# EPICS substitutions: ssaApp/Db/ssa1.substitutions
# asyn record for the underlying asyn octet port
#file "ASYN/db/asynRecord.db" { pattern
#{P,           R,       PORT,      ADDR,   IMAX,    OMAX}
#{SSA1:    OctetAsyn,   ssa1,        0,      125,      123}
#}

# These are the B0 outputs done with bit access.
file "bo_word.template"
{ pattern
{P,           R,        PORT,      OFFSET,   MASK,	ZNAM,  ONAM}
{SSA1:,    OUT1,        RF1_Out_Word,    0,     0x0001,	0, 	1}
{SSA1:,    OUT2,        RF1_Out_Word,    1,     0x0001,	0,	1}
{SSA1:,    OUT4,        RF1_Out_Word,    3,     0x0001,	0,	1}
{SSA1:,    OUT5,        RF1_Out_Word,    4,     0x0001,	0,	1}
{SSA1:,	   OUT6,	RF1_Out_Word,    5,     0x0001,	0,	1}
}

# These are the A0 ouput donw with word write
file "longout.template"
{ pattern
{P,           R,        PORT,      OFFSET}
{SSA1:,    OUT3,        RF1_Out_Word,    2}
}

# There are the Inputs done with bit acess
file "bi_word.template"
{ pattern
{P,           R,        PORT,      OFFSET,   MASK,	ZNAM,  ONAM, 	ZSV, 	OSV, 	 SCAN}
{SSA1:,    BIN1,        RF1_Out_Word,    0,     0x0001,	0, 	1,	NO_ALARM, MAJOR, "I/O Intr"}

}

# There are the Inputs done with word access
file "longin.template"
{ pattern
{P,     R,        PORT,     OFFSET,       SCAN}
{SSA1:,	IN1,	RF1_In_Word,     0,	"I/O Intr"}
{SSA1:, IN2,    RF1_In_Word,     1,      "I/O Intr"}
{SSA1:, IN3,    RF1_In_Word,     2,      "I/O Intr"}
{SSA1:, IN4,    RF1_In_Word,     3,      "I/O Intr"}
{SSA1:, IN5,    RF1_In_Word,     4,      "I/O Intr"}
{SSA1:, IN6,    RF1_In_Word,     5,      "I/O Intr"}
{SSA1:, IN7,    RF1_In_Word,     6,      "I/O Intr"}
{SSA1:, IN8,    RF1_In_Word,     7,      "I/O Intr"}
{SSA1:, IN9,    RF1_In_Word,     8,      "I/O Intr"}
{SSA1:, IN10,   RF1_In_Word,     9,      "I/O Intr"}
{SSA1:, IN11,   RF1_In_Word,     10,     "I/O Intr"}
{SSA1:, IN12,   RF1_In_Word,     11,     "I/O Intr"}
{SSA1:, IN13,   RF1_In_Word,     12,     "I/O Intr"}
{SSA1:, IN14,   RF1_In_Word,     13,     "I/O Intr"}
{SSA1:, IN15,   RF1_In_Word,     14,     "I/O Intr"}
{SSA1:, IN16,   RF1_In_Word,     15,     "I/O Intr"}
{SSA1:, IN17,   RF1_In_Word,     16,     "I/O Intr"}
{SSA1:, IN18,   RF1_In_Word,     17,     "I/O Intr"}
{SSA1:, IN19,   RF1_In_Word,     18,     "I/O Intr"}
{SSA1:, IN20,   RF1_In_Word,     19,     "I/O Intr"}

{SSA1:, IN21,   RF1_In_Word,     20,     "I/O Intr"}
# {SSA1:, IN22,   RF1_In_Word,     21,     "I/O Intr"}
{SSA1:, IN23,   RF1_In_Word,     22,     "I/O Intr"}
{SSA1:, IN24,   RF1_In_Word,     23,     "I/O Intr"}
{SSA1:, IN25,   RF1_In_Word,     24,     "I/O Intr"}
{SSA1:, IN26,   RF1_In_Word,     25,     "I/O Intr"}
{SSA1:, IN27,   RF1_In_Word,     26,     "I/O Intr"}
{SSA1:, IN28,   RF1_In_Word,     27,     "I/O Intr"}
{SSA1:, IN29,   RF1_In_Word,     28,     "I/O Intr"}
{SSA1:, IN30,   RF1_In_Word,     29,     "I/O Intr"}
{SSA1:, IN31,   RF1_In_Word,     30,     "I/O Intr"}
#{SSA1:, IN32,   RF1_In_Word,     31,     "I/O Intr"}
{SSA1:, IN33,   RF1_In_Word,     32,     "I/O Intr"}
#{SSA1:, IN34,   RF1_In_Word,     33,     "I/O Intr"}
{SSA1:, IN35,   RF1_In_Word,     34,     "I/O Intr"}
{SSA1:, IN36,   RF1_In_Word,     35,     "I/O Intr"}
{SSA1:, IN37,   RF1_In_Word,     36,     "I/O Intr"}
{SSA1:, IN38,   RF1_In_Word,     37,     "I/O Intr"}
{SSA1:, IN39,   RF1_In_Word,     38,     "I/O Intr"}
{SSA1:, IN40,   RF1_In_Word,     39,     "I/O Intr"}

{SSA1:, IN41,   RF1_In_Word,     40,     "I/O Intr"}
{SSA1:, IN42,   RF1_In_Word,     41,     "I/O Intr"}
{SSA1:, IN43,   RF1_In_Word,     42,     "I/O Intr"}
#{SSA1:, IN44,   RF1_In_Word,     43,     "I/O Intr"}
#{SSA1:, IN45,   RF1_In_Word,     44,     "I/O Intr"}
#{SSA1:, IN46,   RF1_In_Word,     45,     "I/O Intr"}
{SSA1:, IN47,   RF1_In_Word,     46,     "I/O Intr"}
#{SSA1:, IN48,   RF1_In_Word,     47,     "I/O Intr"}
#{SSA1:, IN49,   RF1_In_Word,     48,     "I/O Intr"}
#{SSA1:, IN50,   RF1_In_Word,     49,     "I/O Intr"}
#{SSA1:, IN51,   RF1_In_Word,     50,     "I/O Intr"}
#{SSA1:, IN52,   RF1_In_Word,     51,     "I/O Intr"}
#{SSA1:, IN53,   RF1_In_Word,     52,     "I/O Intr"}
#{SSA1:, IN54,   RF1_In_Word,     53,     "I/O Intr"}
#{SSA1:, IN55,   RF1_In_Word,     54,     "I/O Intr"}
{SSA1:, IN56,   RF1_In_Word,     55,     "I/O Intr"}
{SSA1:,	IN57,   RF1_In_Word,	56,	"I/O Intr"}
{SSA1:,	IN58,   RF1_In_Word,	57,	"I/O Intr"}
{SSA1:,	IN59,   RF1_In_Word,	58,	"I/O Intr"}
#{SSA1:, IN60,   RF1_In_Word,     59,     "I/O Intr"}

#{SSA1:, IN61,   RF1_In_Word,     60,     "I/O Intr"}
#{SSA1:, IN62,   RF1_In_Word,     61,     "I/O Intr"}
{SSA1:, IN63,   RF1_In_Word,     62,     "I/O Intr"}
#{SSA1:, IN64,   RF1_In_Word,     63,     "I/O Intr"}
#{SSA1:, IN65,   RF1_In_Word,     64,     "I/O Intr"}
#{SSA1:, IN66,   RF1_In_Word,     65,     "I/O Intr"}
#{SSA1:,	IN67,   RF1_In_Word,	66,	"I/O Intr"}
#{SSA1:,	IN68,   RF1_In_Word,	67,	"I/O Intr"}
#{SSA1:,	IN69,   RF1_In_Word,	68,	"I/O Intr"}
#{SSA1:, IN70,   RF1_In_Word,     69,     "I/O Intr"}
#{SSA1:, IN71,   RF1_In_Word,     70,     "I/O Intr"}
{SSA1:, IN72,   RF1_In_Word,     71,     "I/O Intr"}
{SSA1:, IN73,   RF1_In_Word,     72,     "I/O Intr"}
{SSA1:, IN74,   RF1_In_Word,     73,     "I/O Intr"}
{SSA1:, IN75,   RF1_In_Word,     74,     "I/O Intr"}
#{SSA1:, IN76,   RF1_In_Word,     75,     "I/O Intr"}
#{SSA1:,	IN77,   RF1_In_Word,	76,	"I/O Intr"}
#{SSA1:,	IN78,   RF1_In_Word,	77,	"I/O Intr"}
{SSA1:,	IN79,   RF1_In_Word,	78,	"I/O Intr"}
#{SSA1:, IN80,   RF1_In_Word,     79,     "I/O Intr"}

#{SSA1:, IN81,   RF1_In_Word,     80,     "I/O Intr"}
#{SSA1:, IN82,   RF1_In_Word,     81,     "I/O Intr"}
#{SSA1:, IN83,   RF1_In_Word,     82,     "I/O Intr"}
{SSA1:, IN84,   RF1_In_Word,     83,     "I/O Intr"}
{SSA1:, IN85,   RF1_In_Word,     84,     "I/O Intr"}
{SSA1:, IN86,   RF1_In_Word,     85,     "I/O Intr"}
{SSA1:,	IN87,   RF1_In_Word,	86,	"I/O Intr"}
{SSA1:,	IN88,   RF1_In_Word,	87,	"I/O Intr"}
{SSA1:,	IN89,   RF1_In_Word,	88,	"I/O Intr"}
{SSA1:, IN90,   RF1_In_Word,     89,     "I/O Intr"}
{SSA1:, IN91,   RF1_In_Word,     90,     "I/O Intr"}
#{SSA1:, IN92,   RF1_In_Word,     91,     "I/O Intr"}
#{SSA1:, IN93,   RF1_In_Word,     92,     "I/O Intr"}
#{SSA1:, IN94,   RF1_In_Word,     93,     "I/O Intr"}
{SSA1:, IN95,   RF1_In_Word,     94,     "I/O Intr"}
{SSA1:, IN96,   RF1_In_Word,     95,     "I/O Intr"}
{SSA1:,	IN97,   RF1_In_Word,	96,	"I/O Intr"}
#{SSA1:,	IN98,   RF1_In_Word,	97,	"I/O Intr"}
#{SSA1:,	IN99,   RF1_In_Word,	98,	"I/O Intr"}
#{SSA1:,	IN100,  RF1_In_Word,	99,	"I/O Intr"}

#{SSA1:,	IN101,  RF1_In_Word,	100,	"I/O Intr"}
#{SSA1:,	IN102,  RF1_In_Word,	101,	"I/O Intr"}
#{SSA1:,	IN103,  RF1_In_Word,	102,	"I/O Intr"}
{SSA1:,	IN104,  RF1_In_Word,	103,	"I/O Intr"}
{SSA1:,	IN105,  RF1_In_Word,	104,	"I/O Intr"}
{SSA1:,	IN106,  RF1_In_Word,	105,	"I/O Intr"}
{SSA1:,	IN107,  RF1_In_Word,	106,	"I/O Intr"}
{SSA1:,	IN108,  RF1_In_Word,	107,	"I/O Intr"}
{SSA1:,	IN109,  RF1_In_Word,	108,	"I/O Intr"}
{SSA1:,	IN110,  RF1_In_Word,	109,	"I/O Intr"}
{SSA1:,	IN111,  RF1_In_Word,	110,	"I/O Intr"}
{SSA1:,	IN112,  RF1_In_Word,	111,	"I/O Intr"}
{SSA1:,	IN113,  RF1_In_Word,	112,	"I/O Intr"}
{SSA1:,	IN114,  RF1_In_Word,	113,	"I/O Intr"}
{SSA1:,	IN115,  RF1_In_Word,	114,	"I/O Intr"}
{SSA1:,	IN116,  RF1_In_Word,	115,	"I/O Intr"}
}

# These are the aiFloat intput done with read
file "ai.template"
{ pattern
{P,        R,        PORT,      OFFSET,	BITS,   EGUL, EGUF, HOPR, LOPR, PREC, SCAN}
{SSA1:,   IN22,     RF1_In_Word,    21,	0xFFFF,  0,    -0.1, 1e3,  0,  1,   "I/O Intr"}
{SSA1:,   IN32,     RF1_In_Word,    31,	0xFFFF,  0,    -0.1, 1e3,  0,  1,   "I/O Intr"}
{SSA1:,   IN34,     RF1_In_Word,    33,	0xFFFF,  0,    -0.1, 1e3,  0,  1,   "I/O Intr"}
{SSA1:,   IN44,     RF1_In_Word,    43,	0xFFFF,  0,    -0.1, 1e3,  0,  1,   "I/O Intr"}
{SSA1:,   IN45,     RF1_In_Word,    44,	0xFFFF,  0,    -0.1, 1e3,  0,  1,   "I/O Intr"}
{SSA1:,   IN46,     RF1_In_Word,    45,	0xFFFF,  0,    -0.1, 1e3,  0,  1,   "I/O Intr"}
{SSA1:,   IN48,     RF1_In_Word,    47,	0xFFFF,  0,    -0.1, 1e3,  0,  1,   "I/O Intr"}
{SSA1:,   IN49,     RF1_In_Word,    48,	0xFFFF,  0,    -0.1, 1e3,  0,  1,   "I/O Intr"}
{SSA1:,   IN50,     RF1_In_Word,    49,	0xFFFF,  0,    -0.1, 1e3,  0,  1,   "I/O Intr"}
{SSA1:,   IN51,     RF1_In_Word,    50,	0xFFFF,  0,    -0.1, 1e3,  0,  1,   "I/O Intr"}
{SSA1:,   IN52,     RF1_In_Word,    51,	0xFFFF,  0,    -0.1, 1e3,  0,  1,   "I/O Intr"}
{SSA1:,   IN53,     RF1_In_Word,    52,	0xFFFF,  0,    -0.1, 1e3,  0,  1,   "I/O Intr"}
{SSA1:,   IN54,     RF1_In_Word,    53,	0xFFFF,  0,    -0.1, 1e3,  0,  1,   "I/O Intr"}
{SSA1:,   IN55,     RF1_In_Word,    54,	0xFFFF,  0,    -0.1, 1e3,  0,  1,   "I/O Intr"}
{SSA1:,   IN60,     RF1_In_Word,    59,	0xFFFF,  0,    -0.1, 1e3,  0,  1,   "I/O Intr"}
{SSA1:,   IN61,     RF1_In_Word,    60,	0xFFFF,  0,    -0.1, 1e3,  0,  1,   "I/O Intr"}
{SSA1:,   IN62,     RF1_In_Word,    61,	0xFFFF,  0,    -0.1, 1e3,  0,  1,   "I/O Intr"}
{SSA1:,   IN64,     RF1_In_Word,    63,	0xFFFF,  0,    -0.1, 1e3,  0,  1,   "I/O Intr"}
{SSA1:,   IN65,     RF1_In_Word,    64,	0xFFFF,  0,    -0.1, 1e3,  0,  1,   "I/O Intr"}
{SSA1:,   IN66,     RF1_In_Word,    65,	0xFFFF,  0,    -0.1, 1e3,  0,  1,   "I/O Intr"}
{SSA1:,   IN67,     RF1_In_Word,    66,	0xFFFF,  0,    -0.1, 1e3,  0,  1,   "I/O Intr"}
{SSA1:,   IN68,     RF1_In_Word,    67,	0xFFFF,  0,    -0.1, 1e3,  0,  1,   "I/O Intr"}
{SSA1:,   IN69,     RF1_In_Word,    68,	0xFFFF,  0,    -0.1, 1e3,  0,  1,   "I/O Intr"}
{SSA1:,   IN70,     RF1_In_Word,    69,	0xFFFF,  0,    -0.1, 1e3,  0,  1,   "I/O Intr"}
{SSA1:,   IN71,     RF1_In_Word,    70,	0xFFFF,  0,    -0.1, 1e3,  0,  1,   "I/O Intr"}
{SSA1:,   IN76,     RF1_In_Word,    75,	0xFFFF,  0,    -0.1, 1e3,  0,  1,   "I/O Intr"}
{SSA1:,   IN77,     RF1_In_Word,    76,	0xFFFF,  0,    -0.1, 1e3,  0,  1,   "I/O Intr"}
{SSA1:,   IN78,     RF1_In_Word,    77,	0xFFFF,  0,    -0.1, 1e3,  0,  1,   "I/O Intr"}
{SSA1:,   IN80,     RF1_In_Word,    79,	0xFFFF,  0,    -0.1, 1e3,  0,  1,   "I/O Intr"}
{SSA1:,   IN81,     RF1_In_Word,    80,	0xFFFF,  0,    -0.1, 1e3,  0,  1,   "I/O Intr"}
{SSA1:,   IN82,     RF1_In_Word,    81,	0xFFFF,  0,    -0.1, 1e3,  0,  1,   "I/O Intr"}
{SSA1:,   IN83,     RF1_In_Word,    82,	0xFFFF,  0,    -0.1, 1e3,  0,  1,   "I/O Intr"}

{SSA1:,   IN92,     RF1_In_Word,    91,	0xFFFF,  0,    -0.1, 1e3,  0,  1,   "I/O Intr"}
{SSA1:,   IN93,     RF1_In_Word,    92,	0xFFFF,  0,    -0.1, 1e3,  0,  1,   "I/O Intr"}
{SSA1:,   IN94,     RF1_In_Word,    93,	0xFFFF,  0,    -0.1, 1e3,  0,  1,   "I/O Intr"}
{SSA1:,   IN98,     RF1_In_Word,    97,	0xFFFF,  0,    -0.1, 1e3,  0,  1,   "I/O Intr"}
{SSA1:,   IN99,     RF1_In_Word,    98,	0xFFFF,  0,    -0.1, 1e3,  0,  1,   "I/O Intr"}
{SSA1:,   IN100,     RF1_In_Word,   99,	0xFFFF,  0,    -0.1, 1e3,  0,  1,   "I/O Intr"}
{SSA1:,   IN101,     RF1_In_Word,   100,	0xFFFF,  0,    -0.1, 1e3,  0,  1,   "I/O Intr"}
{SSA1:,   IN102,     RF1_In_Word,   101,	0xFFFF,  0,    -0.1, 1e3,  0,  1,   "I/O Intr"}
{SSA1:,   IN103,     RF1_In_Word,   102,	0xFFFF,  0,    -0.1, 1e3,  0,  1,   "I/O Intr"}
}

# Input as intarray
#file "intarray_in.template" { pattern
#{P,	R,		PORT,		NELM,	SCAN}
#{SSA1:,	XnWArray,	RF1_In_Word,	124,	"I/O Intr"}
#}
